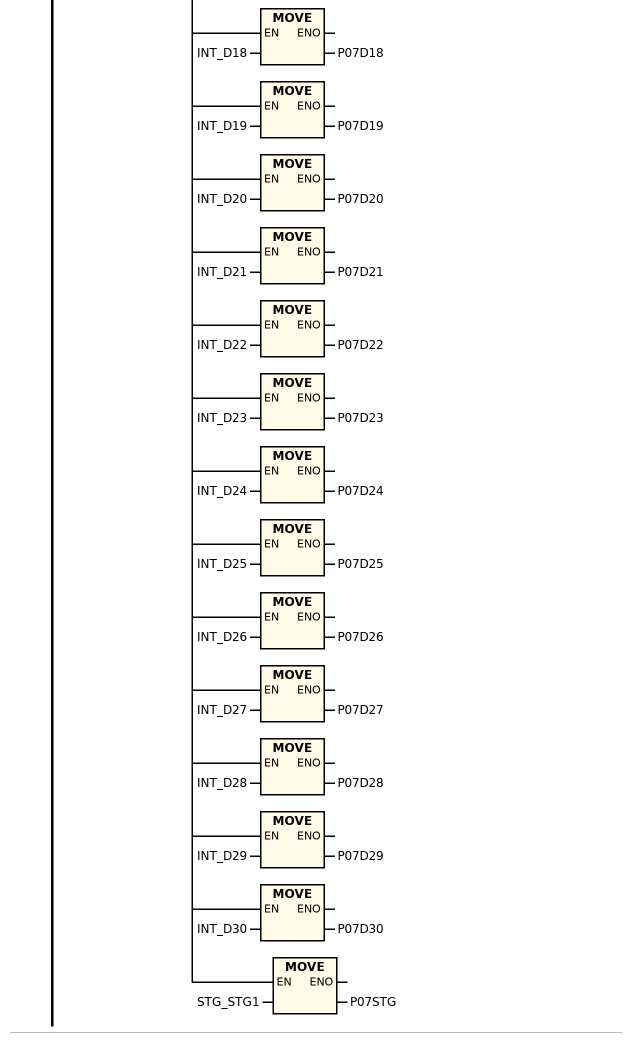
[picture p48: INDIRECT_FN (LD)]
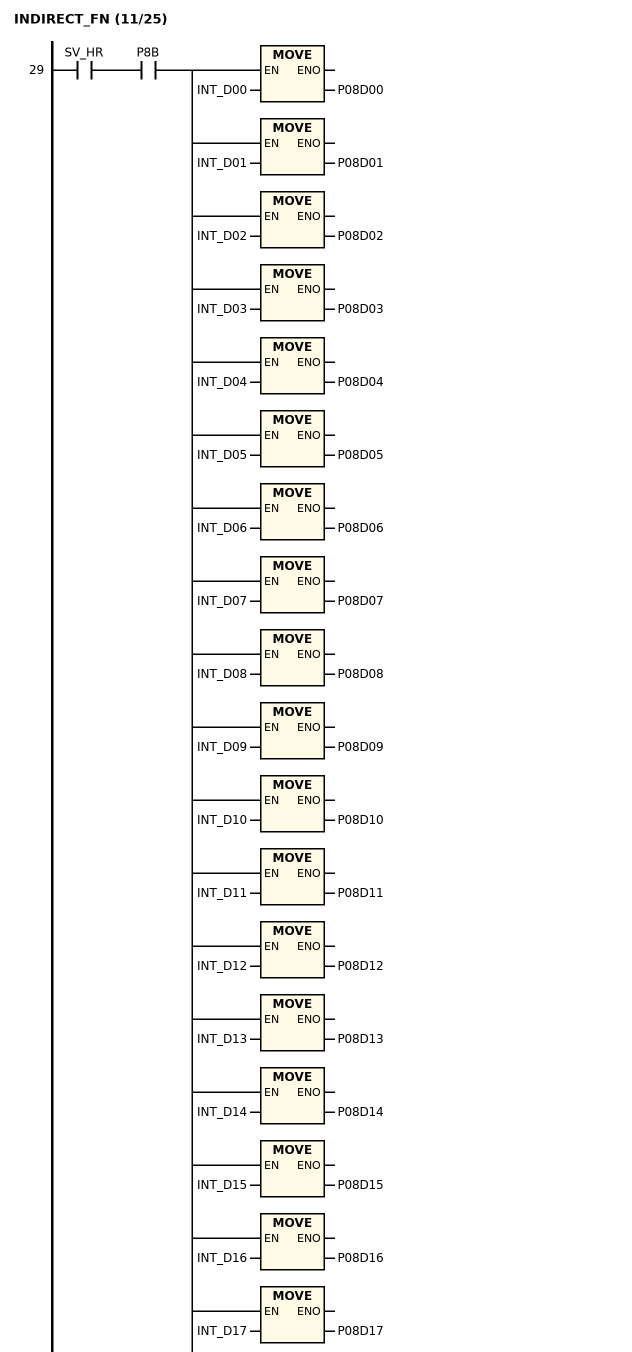
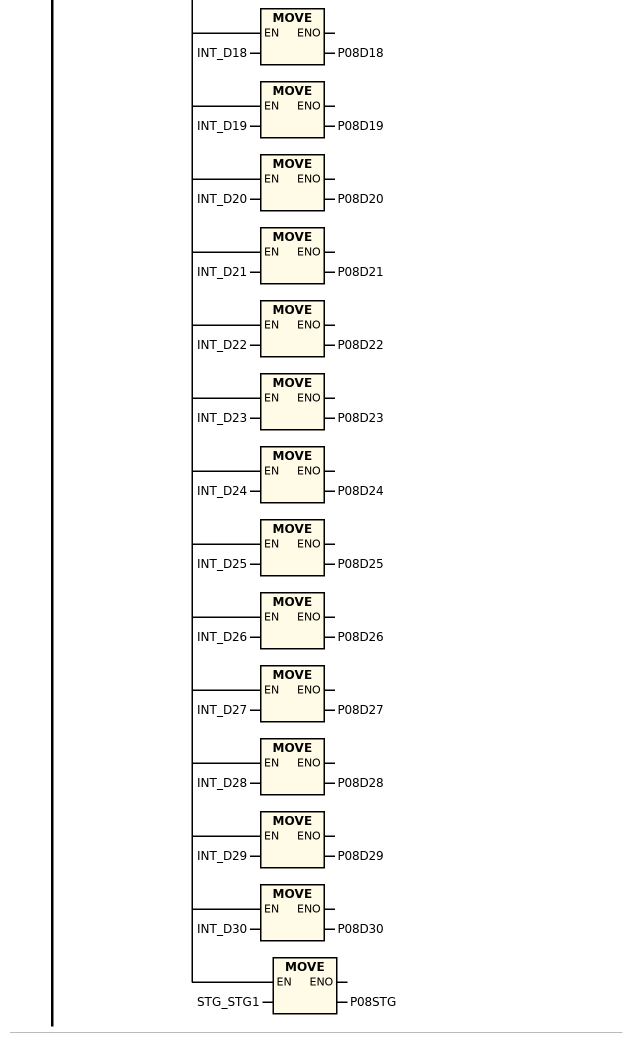
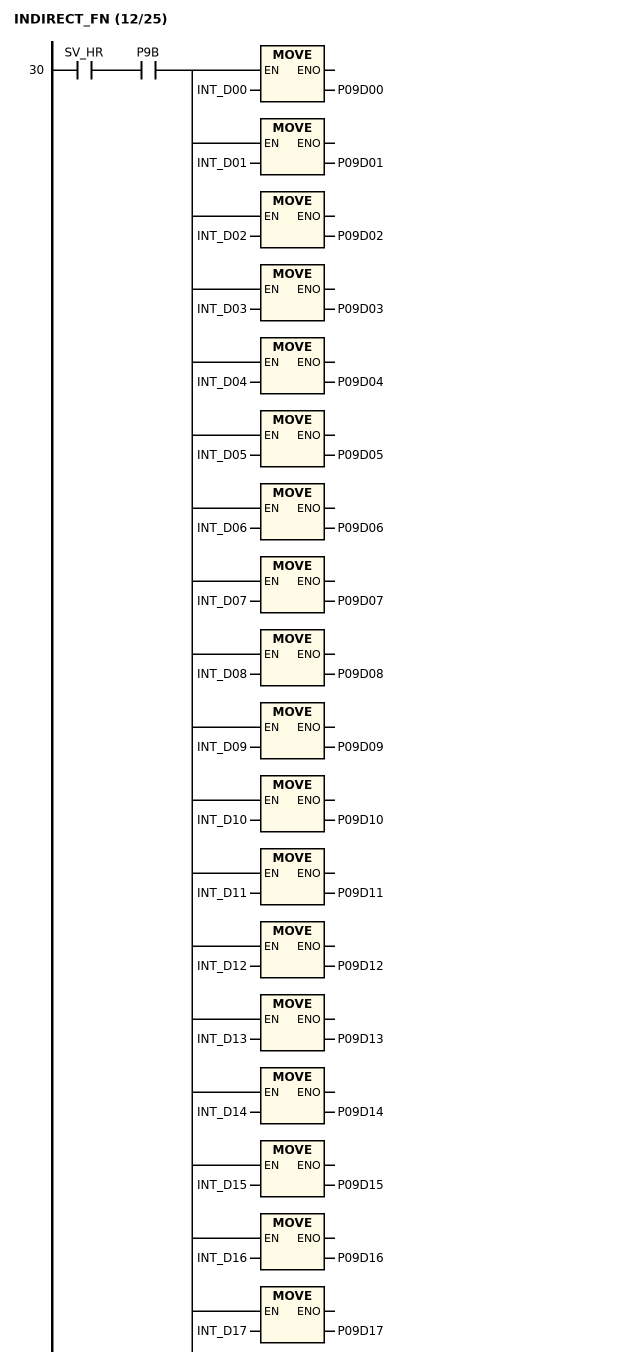
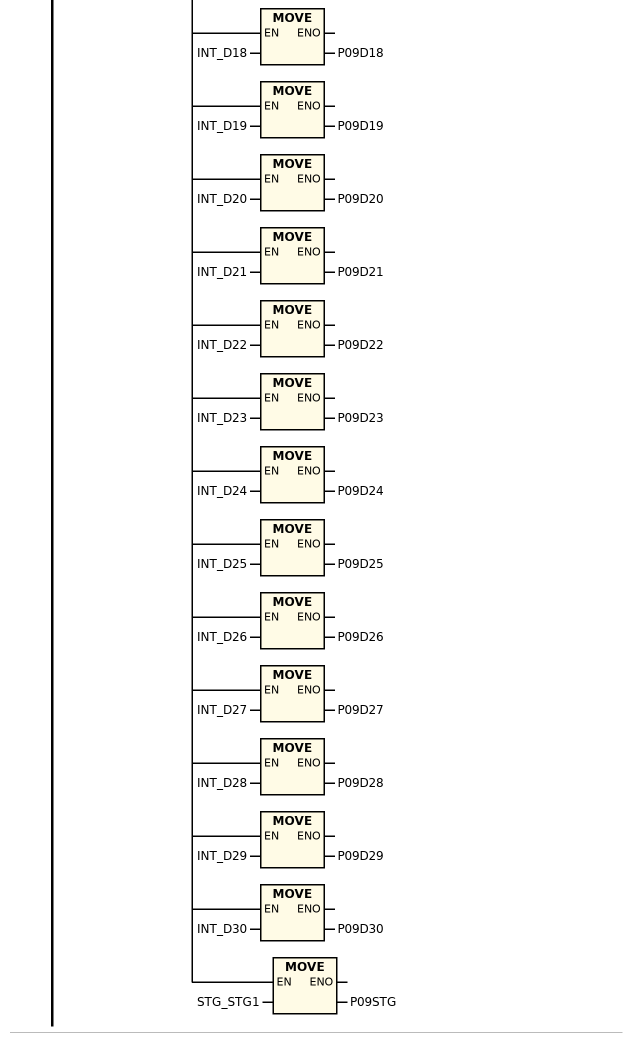
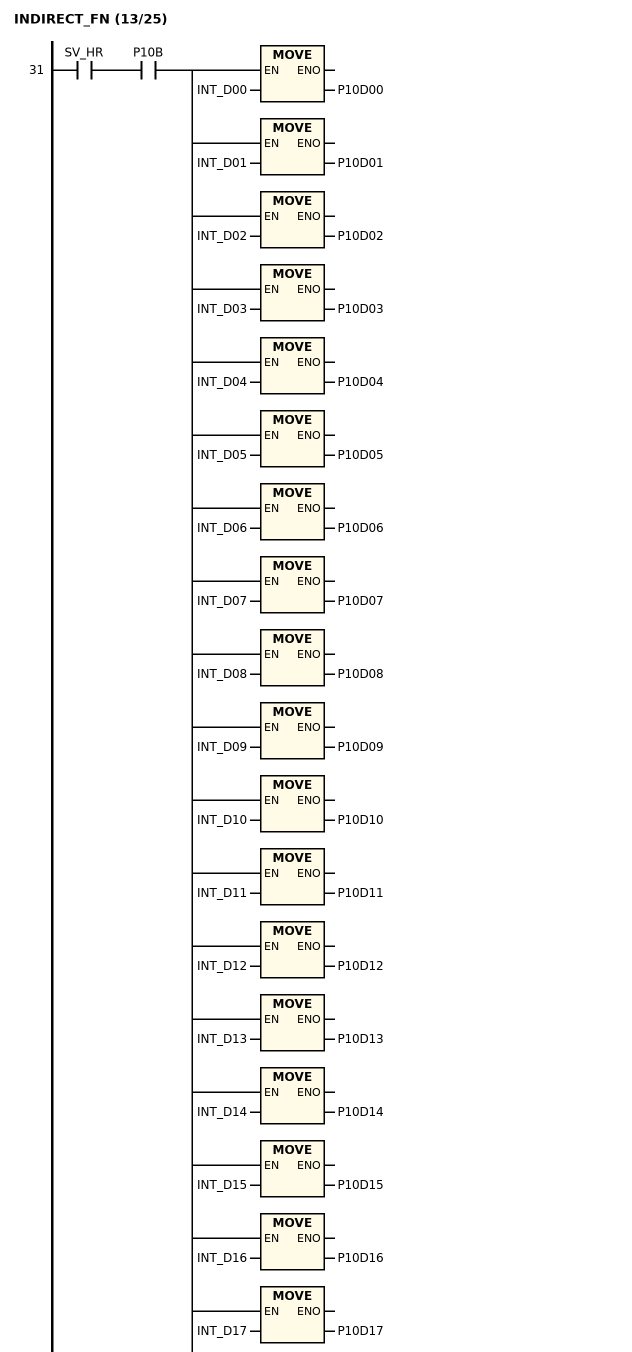
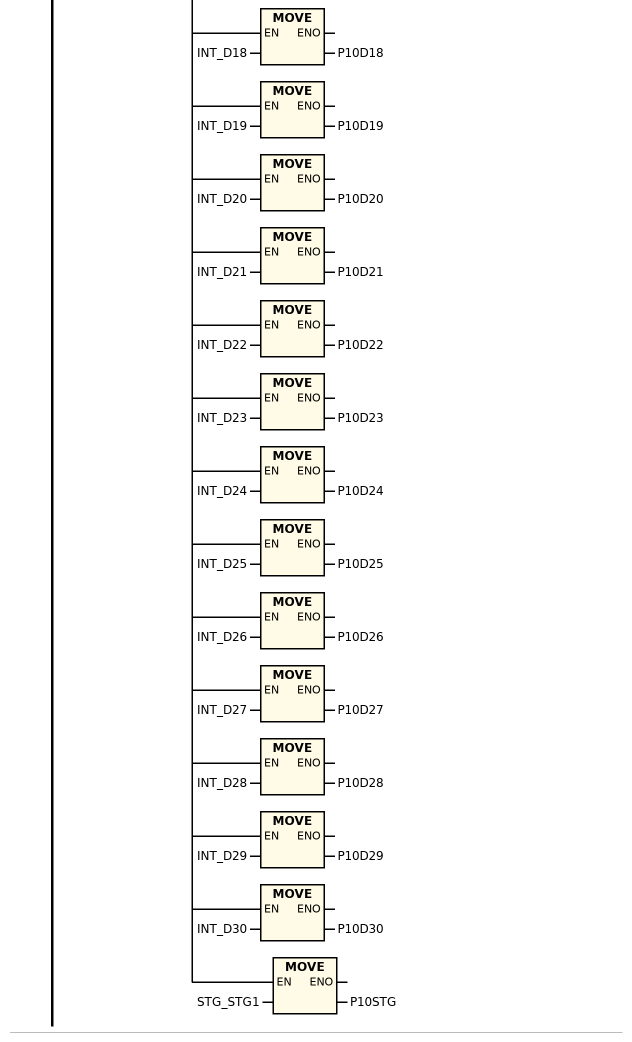
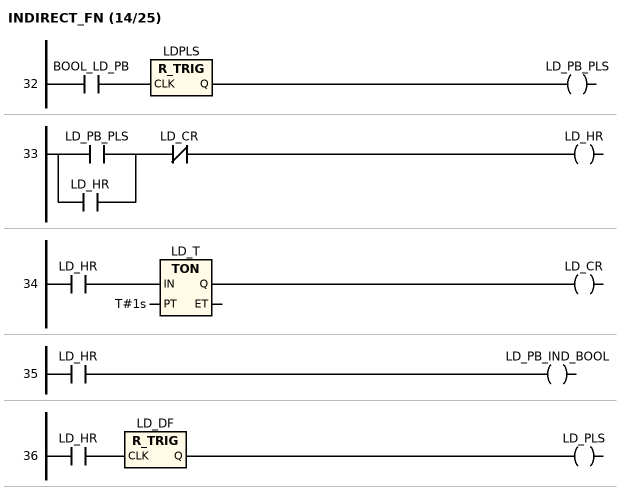
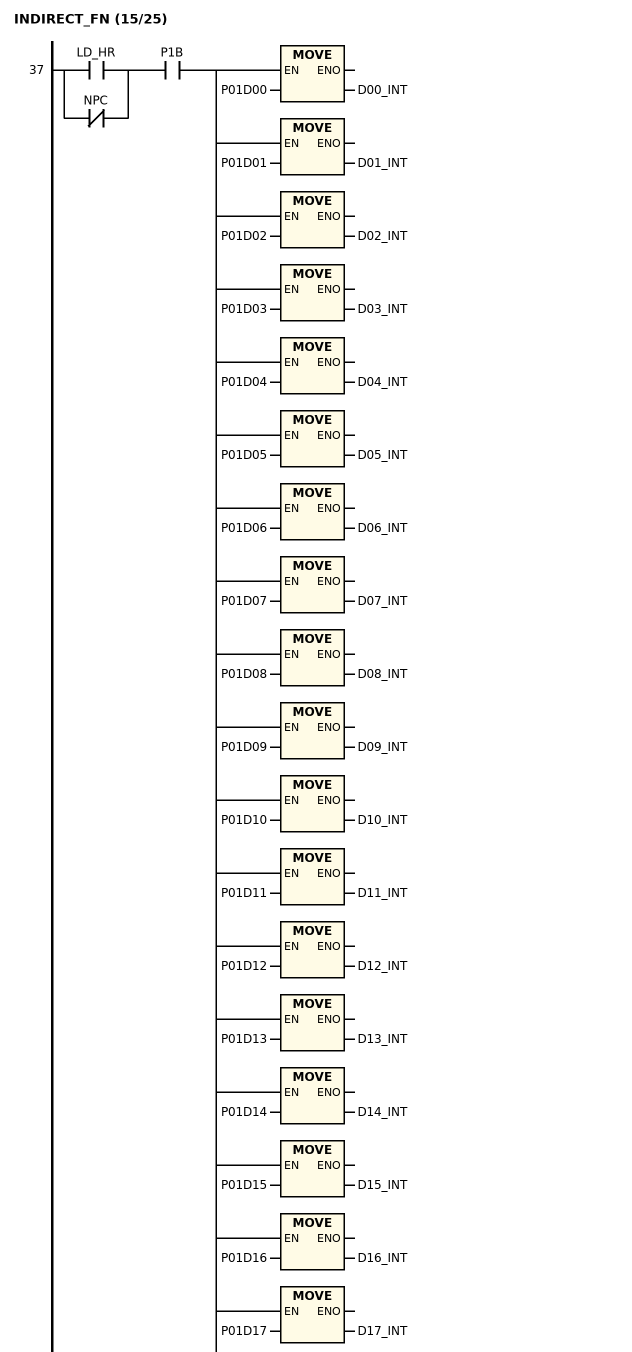
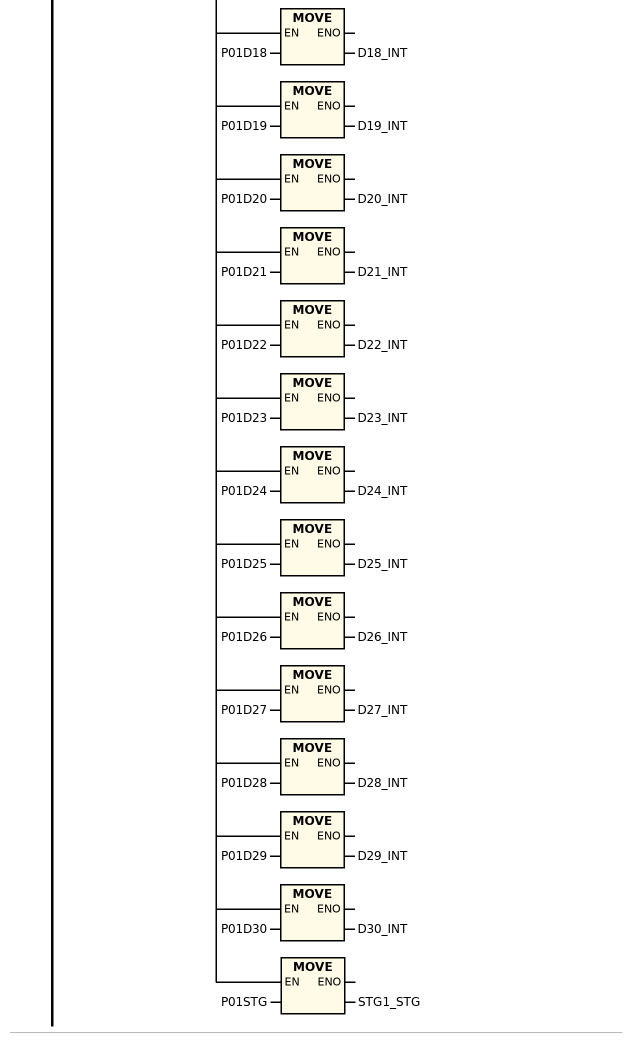
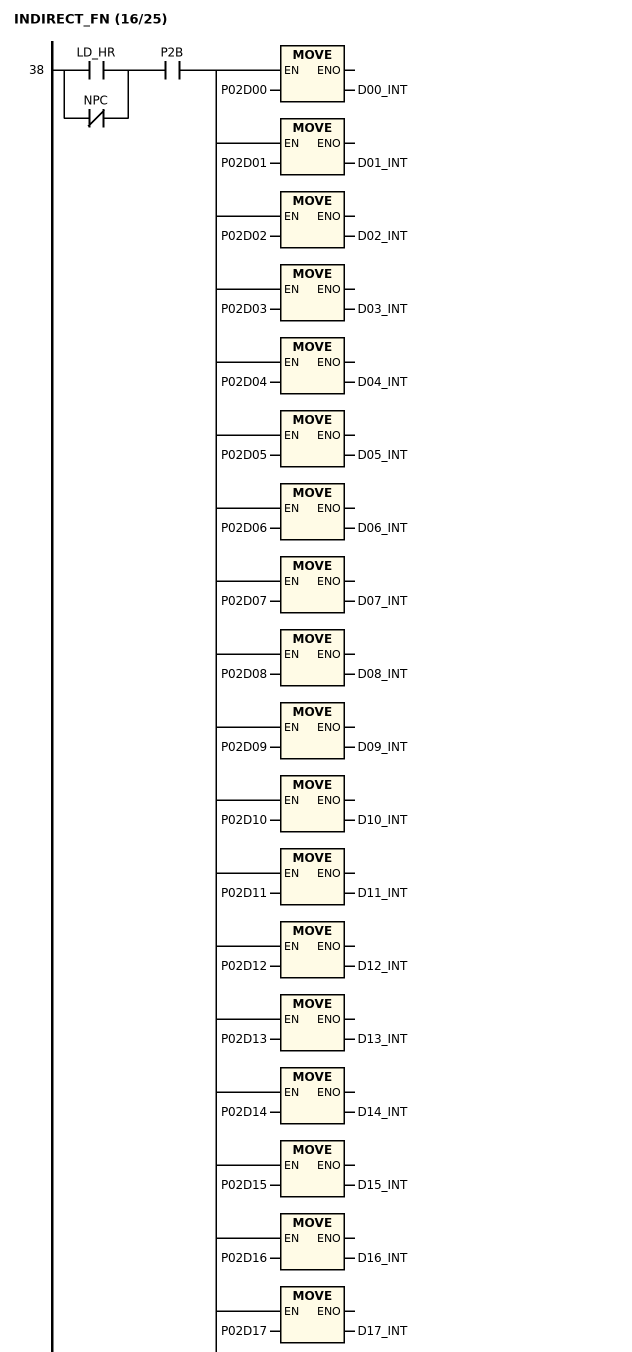
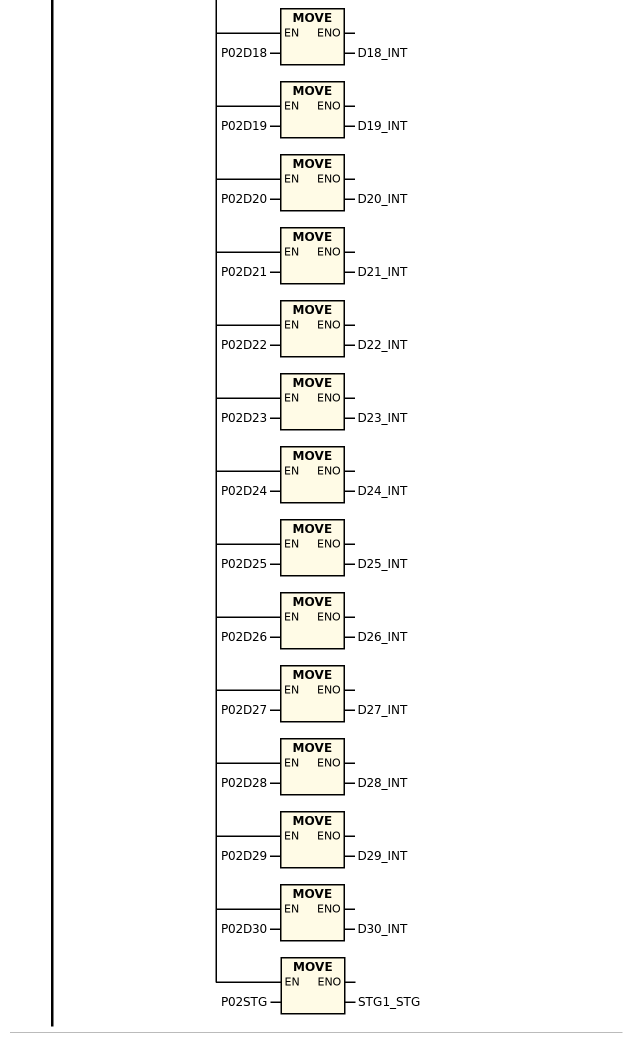
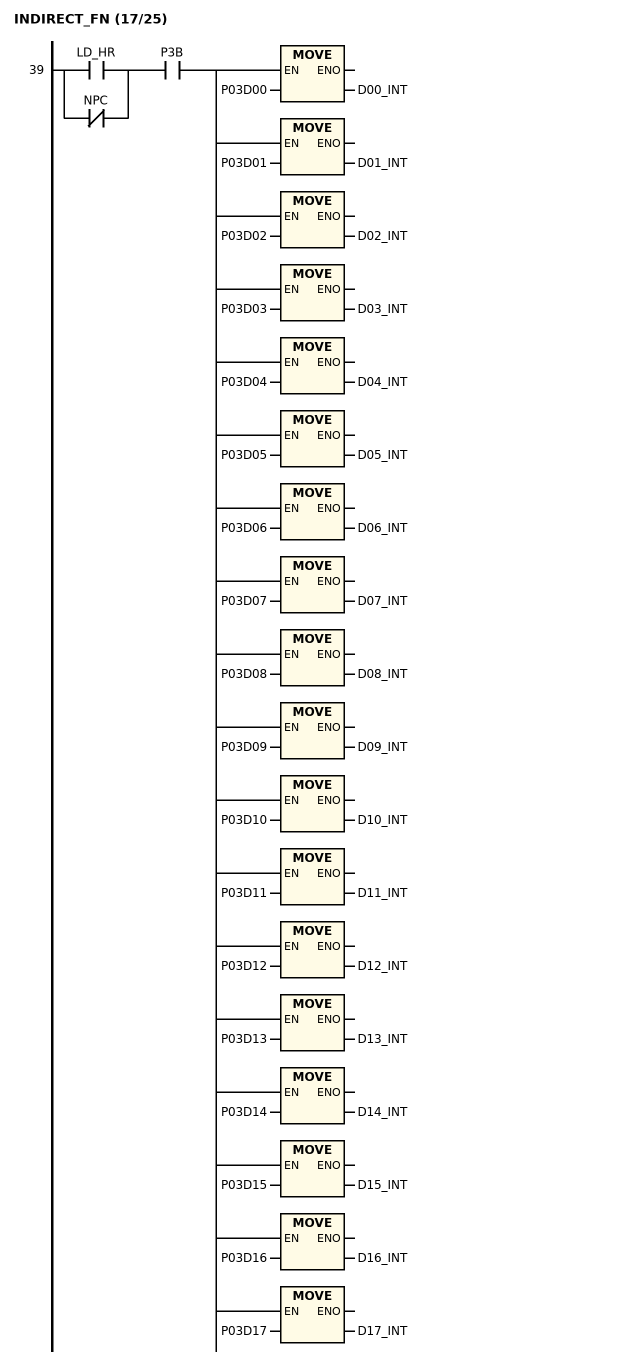
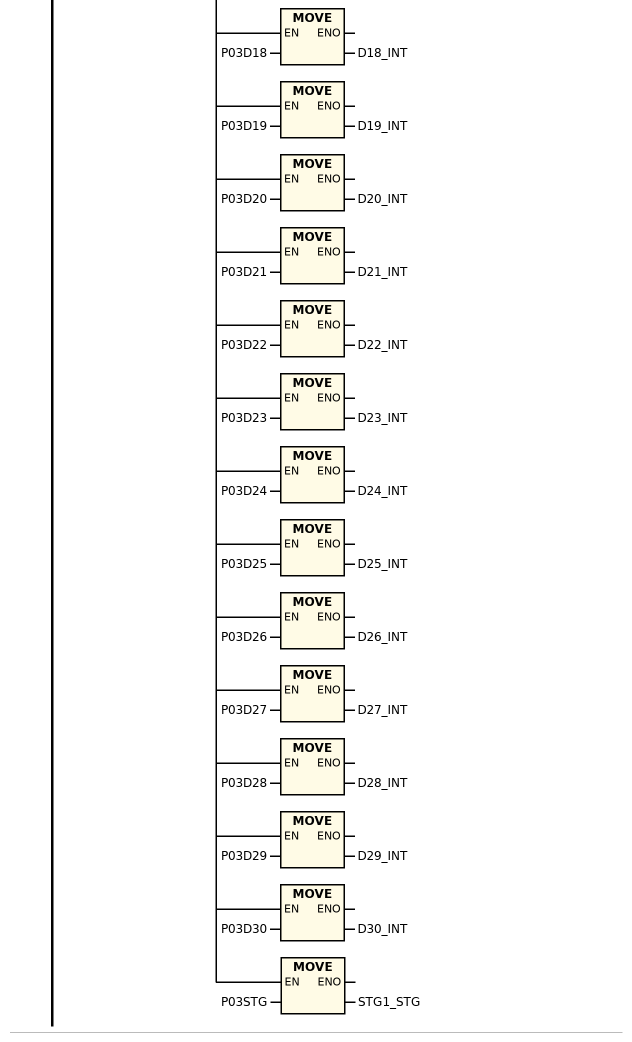
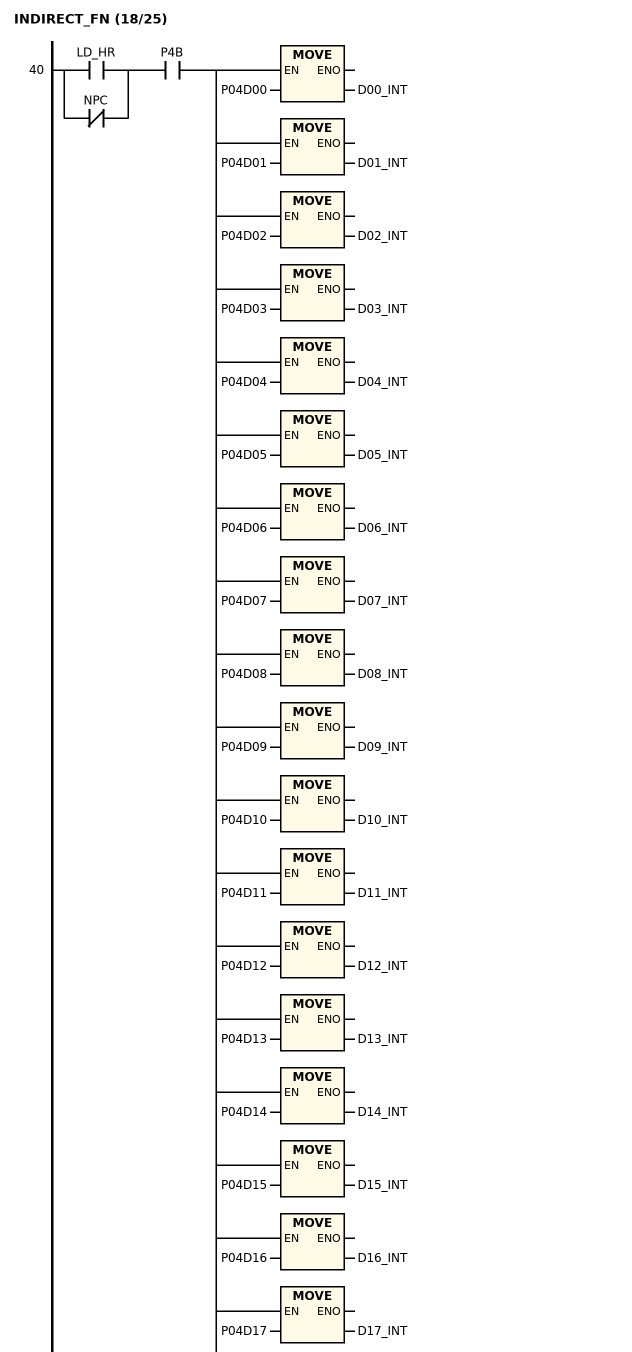
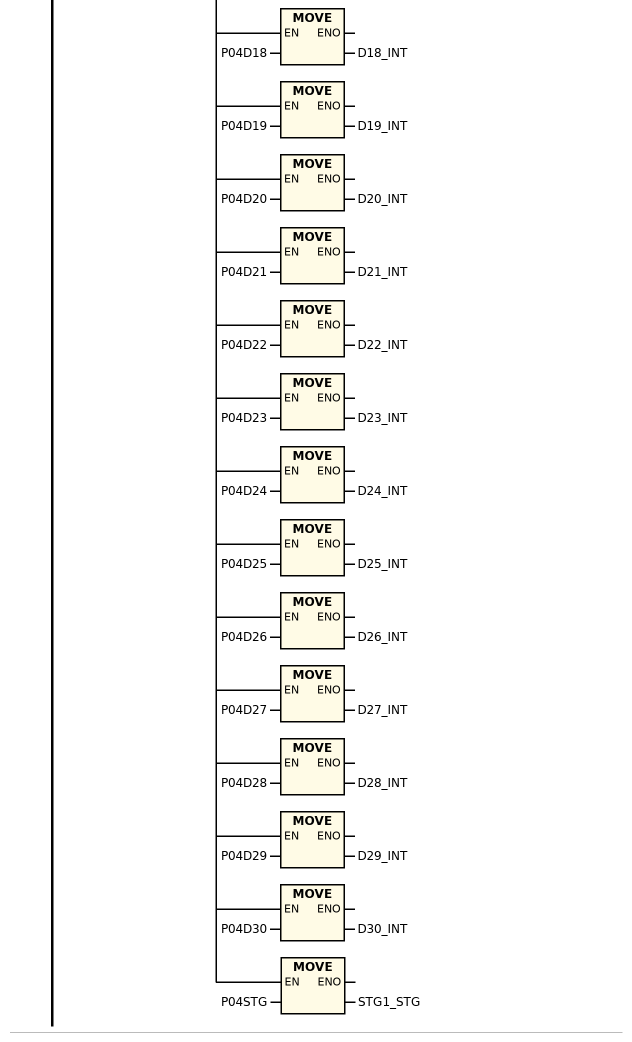
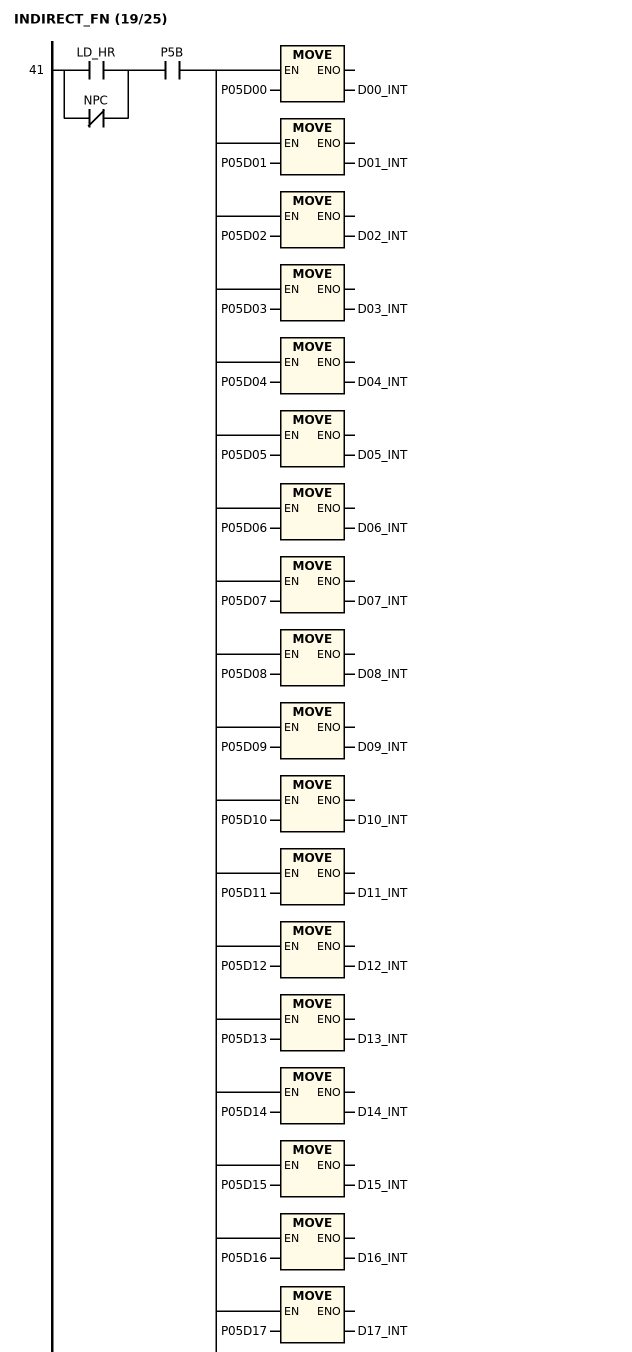
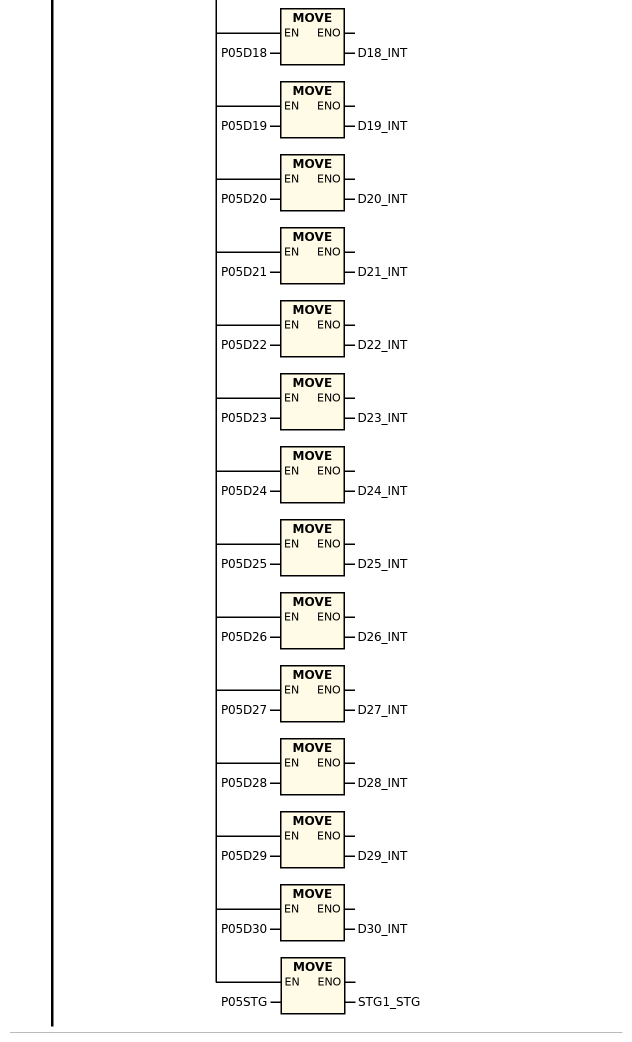
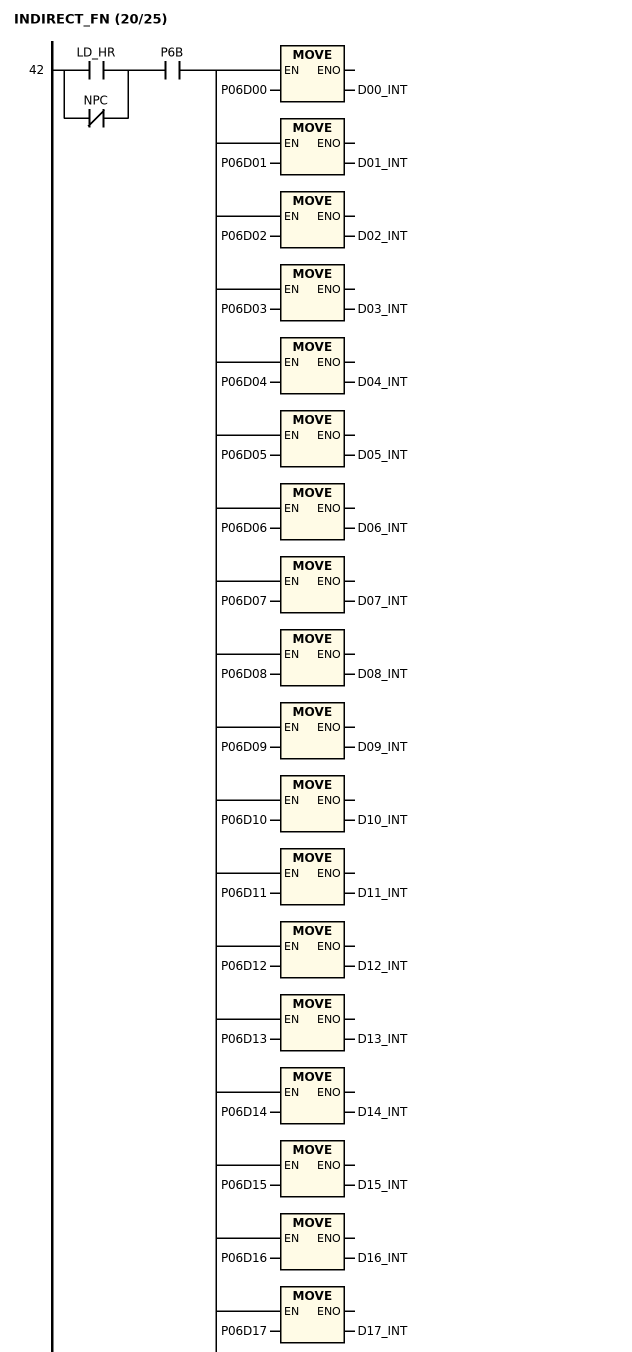
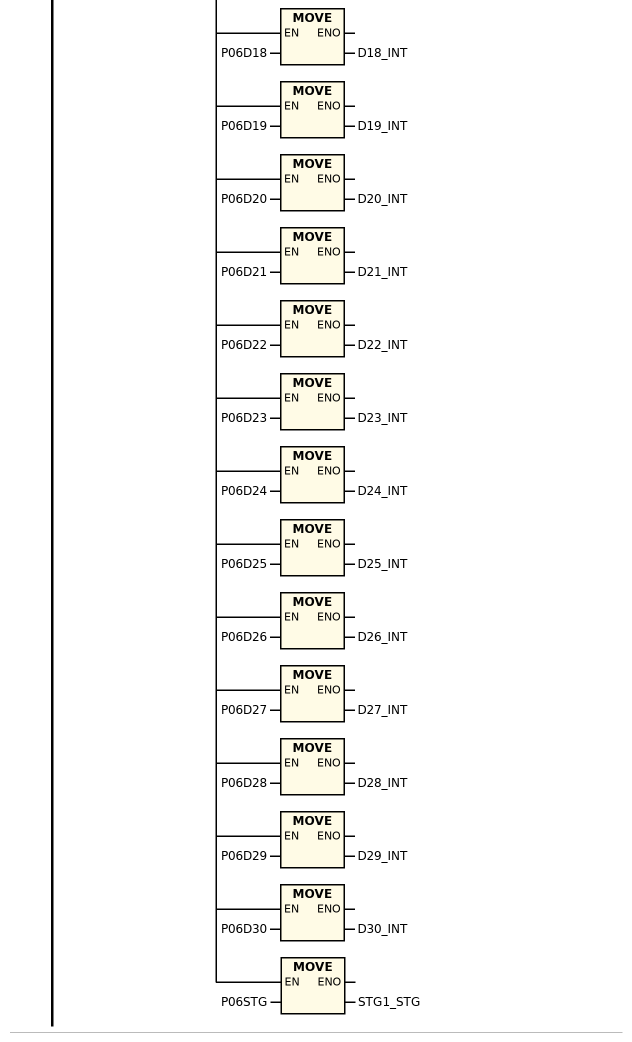
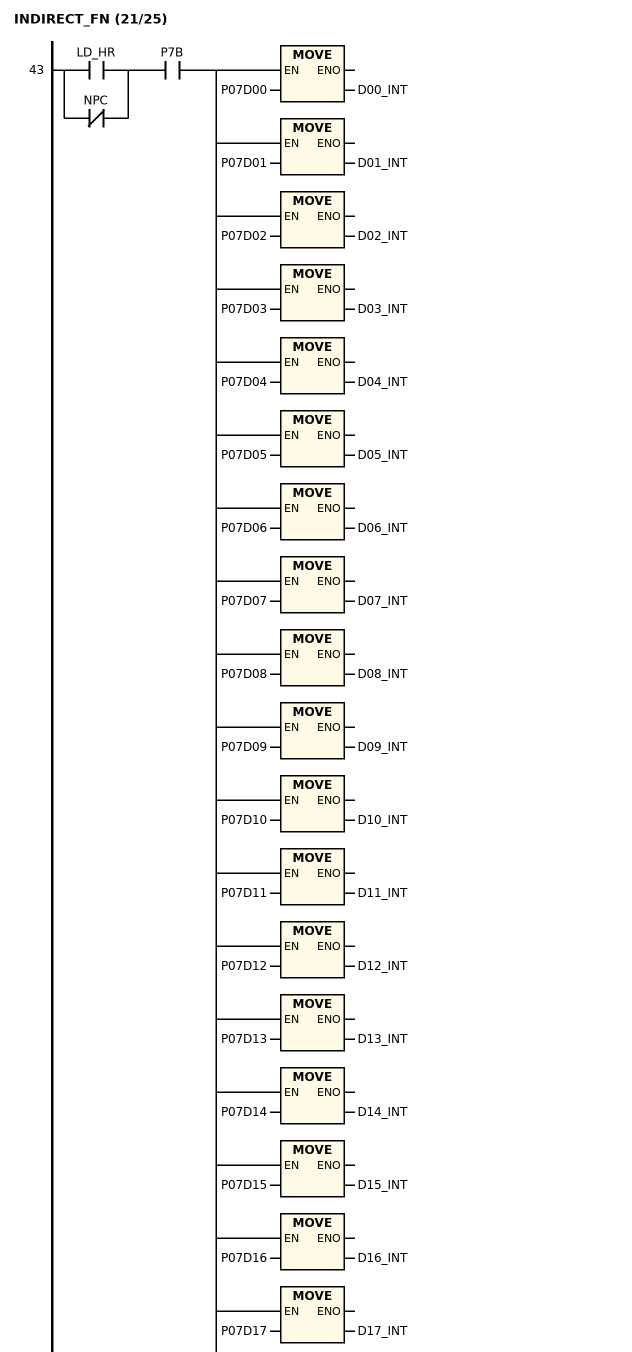
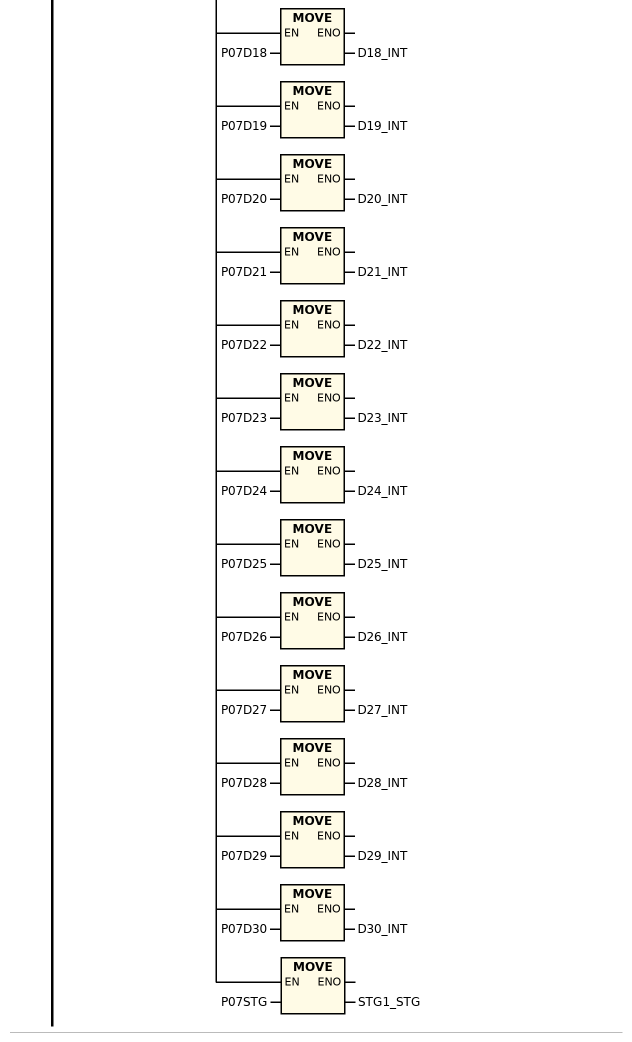
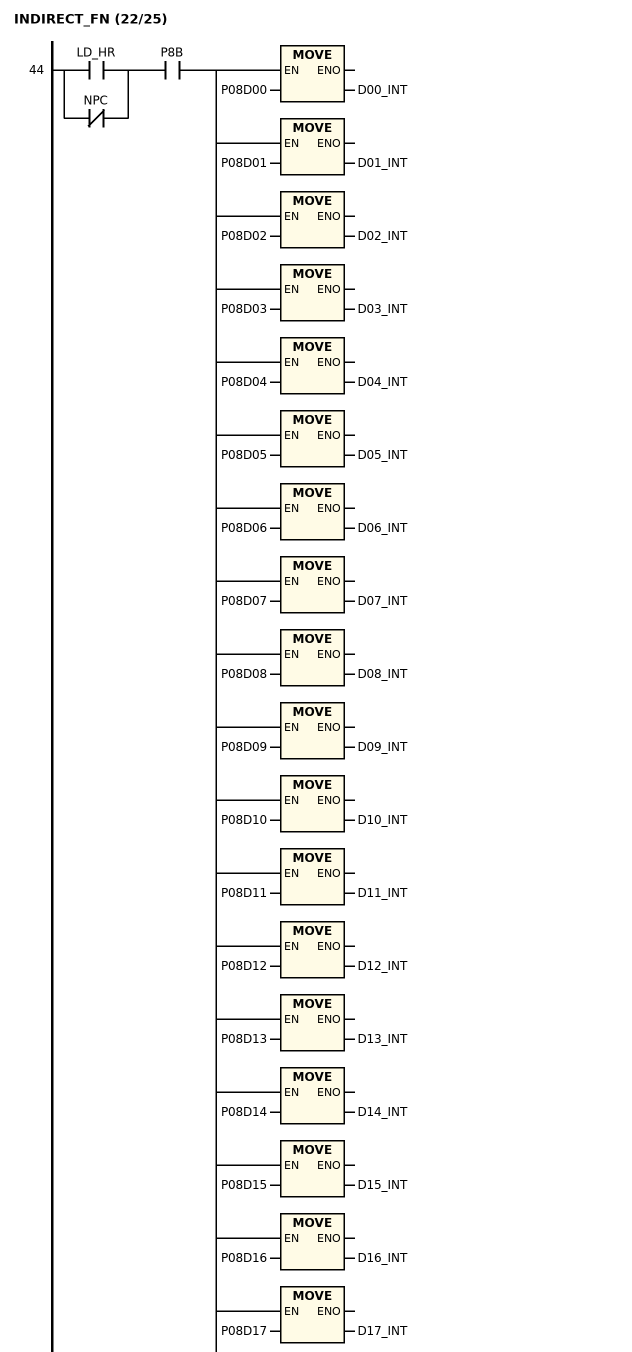
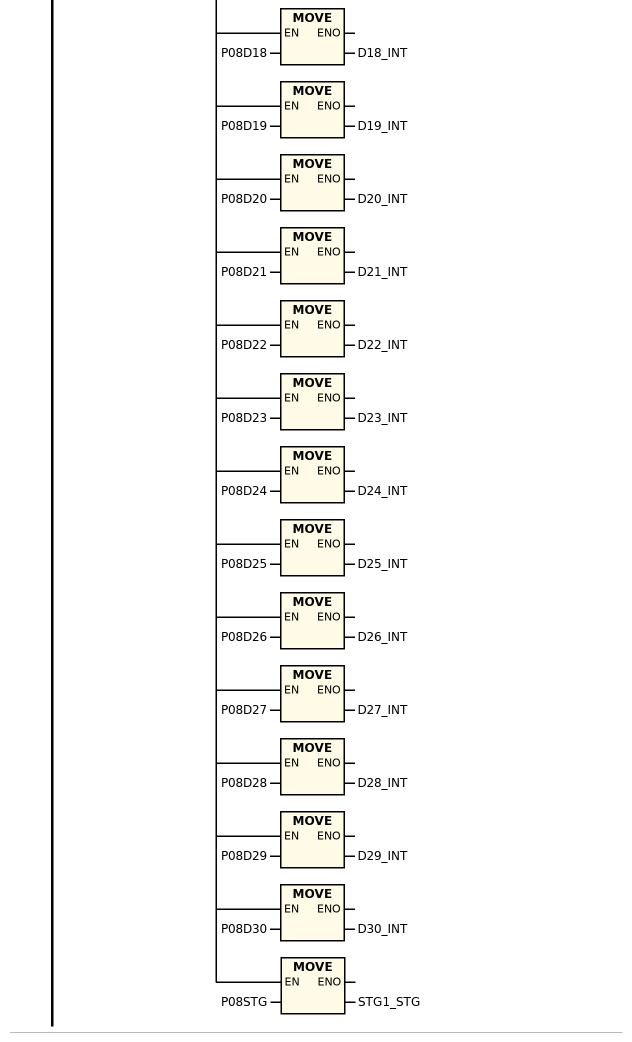
